(* CoDeSys 2.3.8.0 project: TwinCAT NC Sample PTP Move.pro *)
(* Libraries: STANDARD.LIB 5.6.98 12:03:02, TcBase.lib 6.6.06 16:41:28, TcSystem.lib 28.9.07 16:34:46, TcBaseMath.lib 27.7.04 12:07:56, TcMath.lib 23.9.04 15:15:30, TcMC2.lib 26.8.08 09:38:28 *)

(* Task configuration *)
TASK Standard (PRIORITY := 0, INTERVAL := T#10ms);
	MAIN
END_TASK

(* Global variable list: TwinCAT_Configuration *)
(* Generated automatically by TwinCAT - (read only) *)
VAR_CONFIG
	MAIN.Axis1.PlcToNc AT %QB0 : PLCTONC_AXIS_REF;
	MAIN.Axis1.NcToPlc AT %IB0 : NCTOPLC_AXIS_REF;
END_VAR

(* Data type *)
TYPE MoveState_t :
(
	MOVESTATE_INIT,
	MOVESTATE_ENABLE,
	MOVESTATE_FORWARD,
	MOVESTATE_BACKWARDS,
	MOVESTATE_BACKWARDSSLOW,
	MOVESTATE_NEWTARGETPOSITION,
	MOVESTATE_ERROR,
	MOVESTATE_RESET
);
END_TYPE

(* POU MAIN, ST *)
PROGRAM MAIN
VAR
	Axis1 : AXIS_REF;					(* axis reference data structure *)
	state: MoveState_t;				(* state machine state *)

	PowerAxis1: MC_Power;
	PowerAxis1Out: ST_McOutputs;		(* debug function block output data *)

	MoveAxis1: MC_MoveAbsolute;
	MoveAbsoluteOut1: ST_McOutputs;	(* debug function block output data *)

	MoveAxis2: MC_MoveAbsolute;
	MoveAbsoluteOut2: ST_McOutputs;	(* debug function block output data *)

	Reset: MC_Reset;
	ResetOut : ST_McOutputs;			(* debug function block output data *)
END_VAR
	(* update the axis status at the beginning of each cycle *)
	Axis1.ReadStatus;

	(* move axis using a state machine *)
	CASE state OF

		MOVESTATE_INIT :	(* initialisation *)
			(* initialize all function blocks *)
			MoveAxis1.Execute := FALSE;
			MoveAxis2.Execute := FALSE;
			Reset.Execute := FALSE;
			state := MOVESTATE_ENABLE;

		MOVESTATE_ENABLE :
			PowerAxis1.Enable := TRUE;
			PowerAxis1.Enable_Positive := TRUE;
			PowerAxis1.Enable_Negative := TRUE;
			IF PowerAxis1.Status THEN
				state := MOVESTATE_FORWARD;
			ELSIF PowerAxis1.Error THEN
				state := MOVESTATE_ERROR;
			END_IF

		MOVESTATE_FORWARD :		(* start to first position *)
			MoveAxis1.Position := 1500;		(* start to intermediate tartet position *)
			MoveAxis1.Velocity := 500;		(* medium velocity level *)
			MoveAxis1.BufferMode := MC_Buffered;
			MoveAxis1.Execute := TRUE;
			IF MoveAxis1.Active  THEN
				(* axis is executing job but is not yet finished *)
				MoveAxis1.Execute := FALSE;
				(* leave this state and buffer a second command *)
				state := MOVESTATE_NEWTARGETPOSITION;
			ELSIF MoveAxis1.CommandAborted OR MoveAxis1.Error THEN
				state := MOVESTATE_ERROR;
			END_IF

		MOVESTATE_NEWTARGETPOSITION :		(* change target position while moving *)
			(* start a buffered motion command while axis is moving *)
			MoveAxis2.Position := 5000;		(* start to final target *)
			MoveAxis2.Velocity := 1500;		(* increase velocity *)
			MoveAxis2.BufferMode := MC_BlendingPrevious; 	(* use velocity of previous command till intermediate target position position *)
			MoveAxis2.Execute := TRUE;
			IF MoveAxis2.Done THEN
				MoveAxis2.Execute := FALSE;
				state := MOVESTATE_BACKWARDS;
			ELSIF MoveAxis2.CommandAborted OR MoveAxis2.Error THEN
				state := MOVESTATE_ERROR;
			END_IF

		MOVESTATE_BACKWARDS :	(* move back to initial position *)
			MoveAxis1.Position := 100;		(* position close to initial position *)
			MoveAxis1.Velocity := 2000;		(* high velocity *)
			MoveAxis1.BufferMode := MC_Buffered;
			MoveAxis1.Execute := TRUE;
			IF MoveAxis1.Active THEN
				(* axis is executing job but is not yet finished *)
				MoveAxis1.Execute := FALSE;
				(* leave this state and buffer a second command *)
				state := MOVESTATE_BACKWARDSSLOW;
			ELSIF MoveAxis1.CommandAborted OR MoveAxis1.Error THEN
				state := MOVESTATE_ERROR;
			END_IF

		MOVESTATE_BACKWARDSSLOW :	(* move back to initial position *)
			(* start a buffered motion command while axis is moving *)
			MoveAxis2.Position := 0;	(* back to initial position *)
			MoveAxis2.Velocity := 100; 	(* slow velocity *)
			MoveAxis2.BufferMode := MC_BlendingNext; 	(* use velocity from first target position *)
			MoveAxis2.Execute := TRUE;
			IF MoveAxis2.Done THEN
				MoveAxis2.Execute := FALSE;
				state := MOVESTATE_FORWARD;
			ELSIF MoveAxis2.CommandAborted OR MoveAxis2.Error THEN
				state := MOVESTATE_ERROR;
			END_IF

		MOVESTATE_ERROR :
			IF Axis1.Status.Error THEN
				state := MOVESTATE_RESET;	(* axis error requires reset *)
			ELSE
				state := MOVESTATE_INIT;		(* function block errors don't need a reset *)
			END_IF

		MOVESTATE_RESET :
			Reset.Execute := TRUE;
			IF Reset.Done THEN
				state := MOVESTATE_INIT;
			ELSIF Reset.Error THEN
				state := MOVESTATE_INIT; (* can't do anything here *)
			END_IF

	END_CASE

	ActPower;	(* call the power function block *)
	ActMove;	(* call the move function block *)
	ActReset;	(* call the reset function block *)
END_PROGRAM
ACTION ActMove:
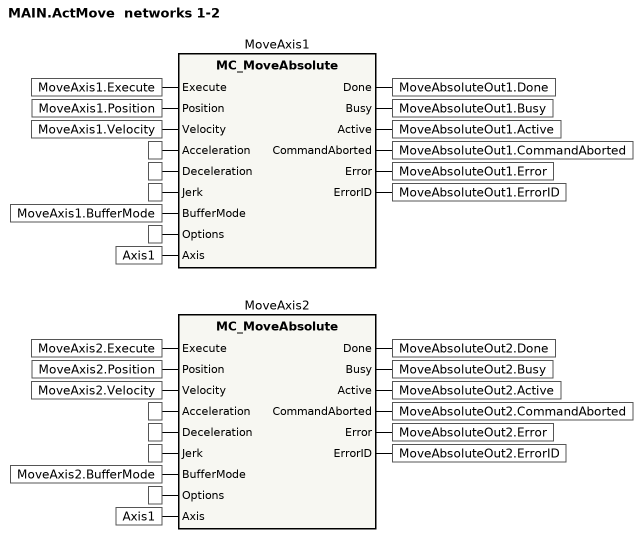
_FBD_ (* Function Block Diagram *)
NETWORK 1
	MoveAxis1:MC_MoveAbsolute(Execute: MoveAxis1.Execute, Position: MoveAxis1.Position, Velocity: MoveAxis1.Velocity, Acceleration: , Deceleration: , Jerk: , BufferMode: MoveAxis1.BufferMode, Options: , Axis: Axis1, Busy => MoveAbsoluteOut1.Busy, Active => MoveAbsoluteOut1.Active, CommandAborted => MoveAbsoluteOut1.CommandAborted, Error => MoveAbsoluteOut1.Error, ErrorID => MoveAbsoluteOut1.ErrorID) => MoveAbsoluteOut1.Done
NETWORK 2
	MoveAxis2:MC_MoveAbsolute(Execute: MoveAxis2.Execute, Position: MoveAxis2.Position, Velocity: MoveAxis2.Velocity, Acceleration: , Deceleration: , Jerk: , BufferMode: MoveAxis2.BufferMode, Options: , Axis: Axis1, Busy => MoveAbsoluteOut2.Busy, Active => MoveAbsoluteOut2.Active, CommandAborted => MoveAbsoluteOut2.CommandAborted, Error => MoveAbsoluteOut2.Error, ErrorID => MoveAbsoluteOut2.ErrorID) => MoveAbsoluteOut2.Done
_END_FBD_
END_ACTION
ACTION ActPower:
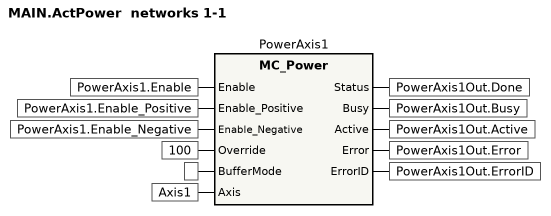
_FBD_ (* Function Block Diagram *)
NETWORK 1
	PowerAxis1:MC_Power(Enable: PowerAxis1.Enable, Enable_Positive: PowerAxis1.Enable_Positive, Enable_Negative: PowerAxis1.Enable_Negative, Override: 100, BufferMode: , Axis: Axis1, Busy => PowerAxis1Out.Busy, Active => PowerAxis1Out.Active, Error => PowerAxis1Out.Error, ErrorID => PowerAxis1Out.ErrorID) => PowerAxis1Out.Done
_END_FBD_
END_ACTION
ACTION ActReset:
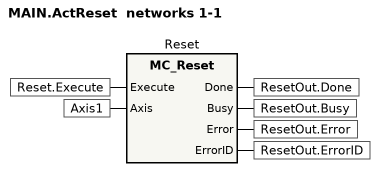
_FBD_ (* Function Block Diagram *)
NETWORK 1
	Reset:MC_Reset(Execute: Reset.Execute, Axis: Axis1, Busy => ResetOut.Busy, Error => ResetOut.Error, ErrorID => ResetOut.ErrorID) => ResetOut.Done
_END_FBD_
(* the same logic as Structured Text *)
(* Network 1 *)
Reset(Execute := Reset.Execute, Axis := Axis1);
ResetOut.Busy := Reset.Busy;
ResetOut.Error := Reset.Error;
ResetOut.ErrorID := Reset.ErrorID;
ResetOut.Done := Reset.Done;
END_ACTION
